{attribute 'qualified_only'}
{attribute 'to_string'}
TYPE ZAppStep :
(
  Undefined := 0
  
  ,BootBegin
  ,BootLoadDefaultData
  ,BootEnd
  ,BootFaultBegin
  ,BootFaultEnd 
  ,RunningBegin
  ,RunningEnd   
);
END_TYPE

(* stored: Version 1.1.0.1
   DUT ZAppStep: Id {afe41ba7-830e-4f70-b90f-ebbff7c2162f} *)
